FUNCTION_BLOCK FB_Draw
VAR
	bDraw			: BOOL;
 	OnTimer 		: TON;
	OffTimer 		: TON;
END_VAR

OnTimer(IN := NOT OffTimer.Q , PT := T#500MS);
OffTimer(IN := OnTimer.Q , PT := T#500ms);
bDraw := OnTimer.Q;

METHOD M_Draw : BOOL
VAR_INPUT
END_VAR
M_Draw := THIS^.bDraw;
END_METHOD

END_FUNCTION_BLOCK

(* stored: Version 1.1.0.1, ProductVersion 3.1.4024.4
   POU FB_Draw: Id {5ce09652-760b-42f0-83d2-cb8b944d73e9}, SpecialFunc None
   Method M_Draw: Id {ac1d1498-a160-4f86-bd37-3831429b1e92} *)
